// TIA Portal V16 export
// export: Created 2021-06-17T11:14:29.7744592Z, ExportSetting WithDefaults, DisplayName Totally Integrated Automation Portal, DisplayVersion V16 Update 4, DisplayName TIA Portal Version Control Interface, DisplayVersion V16 Update 2, DisplayName TIA Portal Openness, DisplayVersion V16 Update 4, DisplayName SINAMICS Startdrive Advanced, DisplayVersion V16 Update 5, DisplayName SINAMICS Startdrive G130, G150, S120, S150, SINAMICS MV, S210, DisplayVersion V16 Update 5, DisplayName SINAMICS Startdrive G110M, G120, G120C, G120D, G120P, G115D, DisplayVersion V16 Update 5, DisplayName STEP 7 Professional, DisplayVersion V16 Update 4, DisplayName SIMATIC Energy Suite, DisplayVersion V16 Update 4, DisplayName STEP 7 Safety, DisplayVersion V16, DisplayName WinCC Advanced / Unified PC, DisplayVersion V16 Update 4, DisplayName SIMATIC Visualization Architect, DisplayVersion V16 Update 1
DATA_BLOCK "RDREC_DB"   // DB8
// stored: AutoNumber true, DBAccessibleFromOPCUA true, InstanceOfName RDREC_SFB, OfSystemLibElement RDREC, OfSystemLibVersion 1.0
"RDREC_SFB"
   // VAR_INPUT
   //    REQ : Bool;
   //    ID : HW_IO;
   //    INDEX : DInt;
   //    MLEN : UInt;
   // END_VAR
   // VAR_OUTPUT
   //    VALID : Bool;
   //    BUSY : Bool;
   //    ERROR : Bool;
   //    STATUS : DWord;
   //    LEN : UInt;
   // END_VAR
   // VAR_IN_OUT
   //    RECORD : Variant;
   // END_VAR
BEGIN
END_DATA_BLOCK
